SYSTEM MGR_TEST (* Test Remote Device Manager Functions *)
  (* Standard: 61499 ITA; Function: Device Manager Functional Test *)
  (* Version 0.0, 2001-11-27, JHC, Rockwell Automation, Copied/Modified from QUERY_TEST. *)
  DEVICE TESTER : FRAME_DEVICE
    RESOURCE RES1 : PANEL_RESOURCE
      FBS
        RQTYPE : IN_CHOICE; (* Request Type Selector *)
        OBJTYPE : IN_CHOICE; (* Object Type Selector *)
        REQUEST : IN_EVENT; (* Generate Request *)
        ARG1 : IN_ANY;
        ARG2 : IN_ANY;
        GEN : RQST_GEN;
        SELTEXT : E_SEL_STRING;
        CLIENT : CLIENT_2_1;
        RTEXT : OUT_TEXT_S;
      END_FBS
      EVENT_CONNECTIONS
        START.COLD TO RQTYPE.INIT;
        START.WARM TO RQTYPE.INIT;
        RQTYPE.INITO TO OBJTYPE.INIT;
        OBJTYPE.INITO TO REQUEST.INIT;
        REQUEST.INITO TO ARG1.INIT;
        ARG1.INITO TO ARG2.INIT;
        ARG2.INITO TO CLIENT.INIT;
        CLIENT.INITO TO RTEXT.INIT;
        REQUEST.IND TO ARG1.REQ;
        ARG1.IND TO ARG2.REQ;
        ARG2.IND TO GEN.REQ;
        GEN.CNF TO SELTEXT.EI0;
        GEN.CNF TO CLIENT.REQ;
        CLIENT.CNF TO SELTEXT.EI1;
        SELTEXT.EO TO RTEXT.REQ;
      END_CONNECTIONS
      DATA_CONNECTIONS
        RQTYPE.OUT TO GEN.RQTYPE;
        OBJTYPE.OUT TO GEN.OBJTYPE;
        ARG1.OUT TO GEN.ARG1;
        ARG2.OUT TO GEN.ARG2;
        GEN.DSTO TO CLIENT.SD_1;
        GEN.RQST TO CLIENT.SD_2;
        GEN.RQST TO SELTEXT.IN0;
        CLIENT.RD_1 TO SELTEXT.IN1;
        SELTEXT.OUT TO RTEXT.IN;
        "FB,Connection" TO OBJTYPE.CHOICES;
        1 TO RQTYPE.QI;
        1 TO OBJTYPE.QI;
        1 TO REQUEST.QI;
        1 TO ARG1.QI;
        1 TO ARG2.QI;
        "REQUEST" TO REQUEST.LABEL;
        1 TO CLIENT.QI;
        "localhost:61494" TO CLIENT.ID;
        "RUT" TO GEN.DSTI;
        1 TO RTEXT.QI;
        "CREATE,DELETE,READ,WRITE,QUERY" TO RQTYPE.CHOICES;
        20 TO ARG1.W;
        "WSTRING" TO ARG1.TYPE;
        "*" TO ARG1.IVAL;
        20 TO ARG2.W;
        "WSTRING" TO ARG2.TYPE;
        "*" TO ARG2.IVAL;
        [8,48] TO RTEXT.SIZE;
      END_CONNECTIONS
    END_RESOURCE
  END_DEVICE
  DEVICE DUT : RMT_FRAME (* Device Under Test *)
    RESOURCE RUT : PANEL_RESOURCE (* Resource Under Test *)
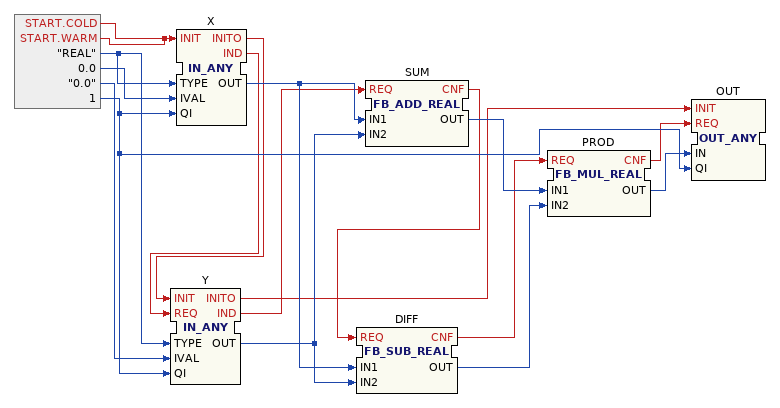
      FBS
        X : IN_ANY;
        Y : IN_ANY;
        SUM : FB_ADD_REAL;
        DIFF : FB_SUB_REAL;
        PROD : FB_MUL_REAL;
        OUT : OUT_ANY; (* X**2-Y**2 *)
      END_FBS
      EVENT_CONNECTIONS
        START.COLD TO X.INIT;
        START.WARM TO X.INIT;
        X.INITO TO Y.INIT;
        Y.INITO TO OUT.INIT;
        X.IND TO Y.REQ;
        Y.IND TO SUM.REQ;
        SUM.CNF TO DIFF.REQ;
        DIFF.CNF TO PROD.REQ;
        PROD.CNF TO OUT.REQ;
      END_CONNECTIONS
      DATA_CONNECTIONS
        X.OUT TO SUM.IN1;
        X.OUT TO DIFF.IN1;
        Y.OUT TO SUM.IN2;
        Y.OUT TO DIFF.IN2;
        SUM.OUT TO PROD.IN1;
        DIFF.OUT TO PROD.IN2;
        PROD.OUT TO OUT.IN;
        "REAL" TO X.TYPE;
        0.0 TO X.IVAL;
        "REAL" TO Y.TYPE;
        "0.0" TO Y.IVAL;
        1 TO X.QI;
        1 TO Y.QI;
        1 TO OUT.QI;
      END_CONNECTIONS
    END_RESOURCE
  END_DEVICE
  DATA_CONNECTIONS (* parameter values *)
    [50,50,375,210] TO TESTER.BOUNDS;
    [1,1] TO TESTER.GRID;
    [425,50,100,150] TO DUT.BOUNDS;
    [1,1] TO DUT.GRID;
    "localhost:61494" TO DUT.MGR_ID;
  END_CONNECTIONS
END_SYSTEM
